// TwinCAT 3 PLC project LeitungszuordnungsTester
// ProgramVersion: 3.1.4022.1
// libraries:
//   Tc2_Standard, * (Beckhoff Automation GmbH)
//   Tc2_System, * (Beckhoff Automation GmbH)
//   Tc3_Module, * (Beckhoff Automation GmbH)
// project tree:
//   / GlobalTextList.TcGTLO, PlcTask.TcTTO (not stored), Visualisierungsmanager.TcVMO (not stored)
//   GVLs/ AN.TcGVL (not stored), DIO.TcGVL (not stored), dSub.TcGVL (not stored), Visu.TcGVL
//   POUs/ LeitungszuordnungsTester.TcPOU, MAIN.TcPOU
//   VISUs/ LeitungszuordnungsTester.TcVIS

// ---- GVLs/Visu.TcGVL
{attribute 'qualified_only'}
VAR_GLOBAL
 NichtVerbunden:BOOL;
 AderErkennen:BOOL;
 Ader_1:BOOL;
 Ader_2:BOOL;
 Ader_3:BOOL;
 Ader_4:BOOL;
 Ader_5:BOOL;
 Ader_6:BOOL;
 Ader_7:BOOL;
 Ader_8:BOOL; 
END_VAR

// ---- POUs/LeitungszuordnungsTester.TcPOU
FUNCTION_BLOCK LeitungszuordnungsTester
VAR_INPUT
END_VAR
VAR_OUTPUT
END_VAR
VAR
END_VAR

IF dio.DI_1 THEN
	Visu.Ader_1:=TRUE;
ELSE 
	Visu.Ader_1 := FALSE;
END_IF

IF dio.DI_2 THEN
	Visu.Ader_2:=TRUE;
ELSE 
	Visu.Ader_2 := FALSE;
END_IF

IF dio.DI_3 THEN
	Visu.Ader_3:=TRUE;
	ELSE 
	Visu.Ader_3 := FALSE;
END_IF

IF dio.DI_4 THEN
	Visu.Ader_4:=TRUE;	
	ELSE 
	Visu.Ader_4 := FALSE;
END_IF

IF dio.DI_5 THEN
	Visu.Ader_5:=TRUE;
	ELSE 
	Visu.Ader_5 := FALSE;
END_IF

IF dio.DI_6 THEN
	Visu.Ader_6:=TRUE;
	ELSE 
	Visu.Ader_6 := FALSE;
END_IF

IF dio.DI_7 THEN
	Visu.Ader_7:=TRUE;
	ELSE 
	Visu.Ader_7 := FALSE;
END_IF

IF dio.DI_8 THEN
	Visu.Ader_8:=TRUE;
	ELSE 
	Visu.Ader_8 := FALSE;
END_IF



IF dio.DI_10 THEN
	Visu.AderErkennen:=TRUE;
	ELSE 
	Visu.AderErkennen := FALSE;
END_IF

IF dio.DI_11 THEN
	Visu.NichtVerbunden:=TRUE;
	ELSE 
	Visu.NichtVerbunden := FALSE;
END_IF

END_FUNCTION_BLOCK

// ---- POUs/MAIN.TcPOU
PROGRAM MAIN
VAR
	LeitungszuordnungsTester: Leitungszuordnungstester;
END_VAR

Leitungszuordnungstester();

END_PROGRAM

// ---- GlobalTextList.TcGTLO
TEXTLIST GlobalTextList
  164 = 'Ader 1 (DQ1)'
  763 = 'Ader 2 (DQ2)'
  940 = 'Ader 3 (DQ3)'
  714 = 'Ader 4 (DQ4)'
  22 = 'Ader 5 (DQ5)'
  514 = 'Ader 6 (DQ6)'
  344 = 'Ader 7 (DQ7)'
  278 = 'Ader 8 (DQ8)'
  648 = 'Ader erkennen ...'
  921 = 'Die zu testende Leitung mit dem Eingang DI1 verbinden'
  394 = 'Leitungszuordnungstester'
  233 = 'Nicht verbunden'
END_TEXTLIST

// ---- VISUs/LeitungszuordnungsTester.TcVIS
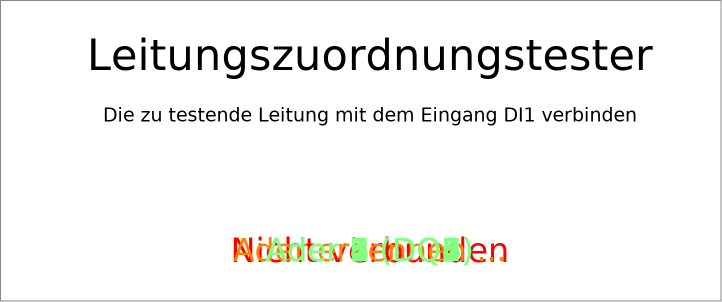
VISUALIZATION LeitungszuordnungsTester  // 722x302
    Label (20,20 700x70), "Leitungszuordnungstester"
    Label (20,100 700x30), "Die zu testende Leitung mit dem Eingang DI1 verbinden"
    Label (20,200 700x100), "Nicht verbunden", invisible if: NOT Visu.NichtVerbunden
    Label (20,200 700x100), "Ader erkennen ...", invisible if: NOT Visu.AderErkennen
    Label (20,200 700x100), "Ader 1 (DQ1)", invisible if: NOT Visu.Ader_1
    Label (20,200 700x100), "Ader 2 (DQ2)", invisible if: NOT Visu.Ader_2
    Label (20,200 700x100), "Ader 3 (DQ3)", invisible if: NOT Visu.Ader_3
    Label (20,200 700x100), "Ader 4 (DQ4)", invisible if: NOT Visu.Ader_4
    Label (20,200 700x100), "Ader 5 (DQ5)", invisible if: NOT Visu.Ader_5
    Label (20,200 700x100), "Ader 6 (DQ6)", invisible if: NOT Visu.Ader_6
    Label (20,200 700x100), "Ader 7 (DQ7)", invisible if: NOT Visu.Ader_7
    Label (20,200 700x100), "Ader 8 (DQ8)", invisible if: NOT Visu.Ader_8
END_VISUALIZATION
